(* CoDeSys 2.3 export: ST_WINCHE_RAMP_CFG.EXP *)

(* Data type *)
TYPE ST_WINCHE_RAMP_CFG :
STRUCT
	Spd_Min : REAL;
	Spd_Inc : REAL;
	Spd_Dec : REAL;
END_STRUCT
END_TYPE
